Staubli VAL3: SENSOR1.dtx

public bool bCalibrating
public bool bTaskDetOK
num nLatchedValue
public num nMaxNumOfObject = 10
public num nNumOfPart = -1
num nObjectID = -1
string sDetNum
string sTASK
trsf trObjectPos
